// TIA Portal project "pidverdaero" (V16)
// Vorlageprojekt für das Buch mit Zielsystem S7-1200

(* hardware
DEVICE "S7-1200-Station_1"  S7-1200 Station
   slot 0: "Baugruppenträger_0"  Rack  V1.0
   slot 1: "PLC_1"  CPU 1211C DC/DC/DC  6ES7 211-1AE40-0XB0  V4.1
   slot 3: "AQ 1x12BIT_1"  AQ1 signal board  6ES7 232-4HA30-0XB0  V1.0
DEVICE "HMI_1"  TP900 Comfort
   slot 0: "HMI_1"  TP900 Comfort  6AV2 124-0JC01-0AX0  16.0.0.0
   slot 1: "HMI_RT_1"  TP900 Comfort  6AV2 124-0JC01-0AX0  16.0.0.0
   slot 5: "HMI_1.IE_CP_1"  PROFINET Interface  16.0.0.0
      slot 1: "Interfaz PROFINET_1"  PROFINET Interface
         slot 1: "Port_1"  Port
         slot 2: "Port_2"  Port
   slot 7: "HMI_1.MPI/DP_CP_1"  MPI/DP Interface  16.0.0.0
*)

// ===== PLC "PLC_1"  CPU 1211C DC/DC/DC =====

VAR_GLOBAL   // PLC tag table "Standard-Variablentabelle"
   "l2" AT %MD40 : Real;
   "l1" AT %MD44 : Real;
   "Kd1" AT %MD0 : Real;
   "Kd2" AT %MD4 : Real;
   "x1e" AT %MD8 : Real;
   "x2e" AT %MD12 : Real;
   "ue" AT %MD16 : Real;
   "u_min" AT %MD20 : Real;
   "u_max" AT %MD24 : Real;
   "z1" AT %MD28 : Real;
   "z2" AT %MD32 : Real;
   "delta_u" AT %MD36 : Real;
   "u_out" AT %MD48 : Real;
   "v1" AT %QD4 : Real;
   "AI_L1" AT %ID4 : Real;
   "AI_L2" AT %ID8 : Real;
   "AO_u" AT %QD0 : Real;
   "x1_hat" AT %MD52 : Real;
   "x2_hat" AT %MD56 : Real;
   "L1_1" AT %MD60 : Real;
   "L1_2" AT %MD64 : Real;
   "L2_1" AT %MD68 : Real;
   "L2_2" AT %MD72 : Real;
   "y1_dev" AT %MD76 : Real;
   "y2_dev" AT %MD80 : Real;
   "x1_hat_dev" AT %MD84 : Real;
   "x2_hat_dev" AT %MD88 : Real;
   "corr1" AT %MD92 : Real;
   "corr2" AT %MD96 : Real;
   "A11" AT %MD100 : Real;
   "A12" AT %MD104 : Real;
   "A21" AT %MD108 : Real;
   "A22" AT %MD112 : Real;
   "B1" AT %MD116 : Real;
   "B2" AT %MD120 : Real;
   "resid1" AT %MD124 : Real;
   "resid2" AT %MD128 : Real;
   "pred1" AT %MD132 : Real;
   "pred2" AT %MD136 : Real;
   "corr_term1" AT %MD140 : Real;
   "corr_term2" AT %MD144 : Real;
   "err1" AT %MD148 : Real;
   "err2" AT %MD152 : Real;
   "start" AT %I60.0 : Bool;
   "pid11" AT %Q8.0 : Bool;
   "pid22" AT %Q8.1 : Bool;
   "Kp" AT %MD156 : Real;
   "Ki" AT %MD160 : Real;
   "Kd" AT %MD164 : Real;
   "Ts" AT %MD168 : Real;
   "SetPoint" AT %MD172 : Real;
   "error" AT %MD176 : Real;
   "P_term" AT %MD180 : Real;
   "I_term" AT %MD184 : Real;
   "I_prev" AT %MD188 : Real;
   "D_term" AT %MD192 : Real;
   "error_prev" AT %MD196 : Real;
   "u_raw" AT %MD200 : Real;
END_VAR

DATA_BLOCK "OnOff_DB"   // DB2
{ S7_Optimized_Access := 'TRUE' }
VERSION : 0.1
// stored: InstanceOfName OnOff
"OnOff"
BEGIN
END_DATA_BLOCK

DATA_BLOCK "OnOff_DB2"   // DB4
{ S7_Optimized_Access := 'TRUE' }
VERSION : 0.1
// stored: InstanceOfName OnOff
"OnOff"
BEGIN
END_DATA_BLOCK

DATA_BLOCK "OnOff_DB_1"   // DB5
{ S7_Optimized_Access := 'TRUE' }
VERSION : 0.1
// stored: InstanceOfName OnOff
"OnOff"
BEGIN
END_DATA_BLOCK

DATA_BLOCK "I"   // DB6
{ S7_Optimized_Access := 'TRUE' }
VERSION : 0.1
// stored: InstanceOfName lqg1
"lqg1"
BEGIN
END_DATA_BLOCK

// folder: System blocks/Program resources

DATA_BLOCK "IEC_Timer_0_DB"   // DB1
{ S7_Optimized_Access := 'TRUE' }
AUTHOR : Simatic
FAMILY : IEC
NAME : IEC_TMR
VERSION : 1.0
// stored: InstanceOfName IEC_TIMER
"IEC_TIMER"
BEGIN
END_DATA_BLOCK

// folder: (top level)

FUNCTION_BLOCK "OnOff"   // FB1, SCL
{ S7_Optimized_Access := 'TRUE' }
VERSION : 0.1
BEGIN
   // ==============================
   // 0) PARÁMETROS PID (BALANCEADO)
   // ==============================
   // Ganancias calculadas con pidtune (Robustez 60deg)
   "Kp" := 2.9222;
   "Ki" := 0.0231;
   "Kd" := 32.0832;

   // Tiempo de muestreo (Debe ser igual al Cyclic Interrupt, ej. 0.05s)
   "Ts" := 0.05;

   // Referencia (Set Point) - A donde quieres que llegue el agua
   "SetPoint" := 2.0;

   // Límites del Actuador
   "u_min" := 0.0;
   "u_max" := 10.0;

   // ==============================
   // 1) LECTURA Y ESCALADO (IGUAL AL LQG)
   // ==============================

   "l1" := ("l1" * 0.9) + (("AI_L1" * 0.3) * 0.1);
   "l2" := "AI_L2" * 0.3;

   // Cálculo de caudal (Solo para monitoreo)
   "v1" := 4.073 * SQRT("l2");

   // ==============================
   // 2) CÁLCULO DEL ERROR
   // ==============================

   // Error actual = Lo que quiero - Lo que tengo
   "error" := "SetPoint" - "l1";

   // ==============================
   // 3) ALGORITMO PID
   // ==============================

   // --- TÉRMINO PROPORCIONAL (P) ---
   "P_term" := "Kp" * "error";

   // --- TÉRMINO INTEGRAL (I) ---
   // Acumula el error: I_nuevo = I_viejo + (Ki * error * Tiempo)
   // "I_prev" debe ser variable STATIC (Memoria)
   "I_term" := "I_prev" + ("Ki" * "error" * "Ts");

   // --- TÉRMINO DERIVATIVO (D) ---
   // Velocidad del error: D = Kd * (error - error_anterior) / Tiempo
   // "error_prev" debe ser variable STATIC (Memoria)
   "D_term" := "Kd" * ("error" - "error_prev") / "Ts";

   // --- SUMA TOTAL ---
   "u_raw" := "P_term" + "I_term" + "D_term";

   // ==============================
   // 4) SATURACIÓN Y ANTI-WINDUP
   // ==============================

   IF "u_raw" > "u_max" THEN
       "u_out" := "u_max";
       "I_term" := "I_prev"; // Congelar Integral

   ELSIF "u_raw" < "u_min" THEN
       "u_out" := "u_min";
       "I_term" := "I_prev"; // Congelar Integral

   ELSE
       "u_out" := "u_raw";
       "I_prev" := "I_term"; // Guardar Integral nueva
   END_IF;

   // ==============================
   // 5) ACTUALIZACIÓN DE MEMORIAS
   // ==============================
   // Guardamos el error actual para usarlo como "pasado" en el siguiente ciclo
   "error_prev" := "error";

   // ==============================
   // 6) SALIDA AL ACTUADOR
   // ==============================
   "AO_u" := "u_out";
END_FUNCTION_BLOCK

FUNCTION_BLOCK "lqg1"   // FB2, SCL
{ S7_Optimized_Access := 'TRUE' }
VERSION : 0.1
BEGIN
   // ==========================================
   // 1. PARÁMETROS (Tus Ganancias Altas)
   // ==========================================
   "Kp" := 4.1326;
   "Ki" := 0.0461;
   "Kd" := 82.0658;

   "Ts" := 0.05;      // Tiempo de ciclo
   "SetPoint" := 1.0; // Referencia (1 metro)
   "u_min" := 0.0;
   "u_max" := 10.0;

   // ==========================================
   // 2. LECTURA Y FILTRO (EN UNA SOLA LÍNEA)
   // ==========================================

   // Truco: Usamos "l1" para guardar el valor filtrado. 
   // 0.9 = Memoria (Suavidad) | 0.1 = Lectura Nueva (Sensor)
   // ESTO ELIMINA EL RUIDO SIN CREAR VARIABLES NUEVAS
   "l1" := ("l1" * 0.9) + (("AI_L1" * 0.3) * 0.1);

   // Lectura Tanque 2 (Solo visual, sin filtro)
   "l2" := "AI_L2" * 0.3;
   "v1" := 4.073 * SQRT("l2");

   // ==========================================
   // 3. CÁLCULO DEL ERROR
   // ==========================================
   "error" := "SetPoint" - "l1";

   // ==========================================
   // 4. ALGORITMO PID (ESTÁNDAR)
   // ==========================================

   // -- PROPORCIONAL --
   "P_term" := "Kp" * "error";

   // -- INTEGRAL (ACUMULATIVA) --
   // "I_prev" DEBE SER STATIC (Memoria)
   "I_term" := "I_prev" + ("Ki" * "error" * "Ts");

   // -- DERIVATIVO (VELOCIDAD) --
   // "error_prev" DEBE SER STATIC (Memoria)
   "D_term" := "Kd" * ("error" - "error_prev") / "Ts";

   // -- SUMA TOTAL --
   "u_raw" := "P_term" + "I_term" + "D_term";

   // ==========================================
   // 5. SATURACIÓN Y ANTI-WINDUP
   // ==========================================

   IF "u_raw" > "u_max" THEN
       "u_out" := "u_max";
       "I_term" := "I_prev"; // Congelar Integral

   ELSIF "u_raw" < "u_min" THEN
       "u_out" := "u_min";
       "I_term" := "I_prev"; // Congelar Integral

   ELSE
       "u_out" := "u_raw";
       "I_prev" := "I_term"; // Guardar Integral nueva
   END_IF;

   // ==========================================
   // 6. GUARDAR MEMORIA
   // ==========================================
   "error_prev" := "error"; // Guardar error para la derivada del siguiente ciclo

   // ==========================================
   // 7. SALIDA FÍSICA
   // ==========================================
   "AO_u" := "u_out";
END_FUNCTION_BLOCK

FUNCTION "MHJ-PLC-Lab-Function-S71200" : Void   // FC9000, SCL
{ S7_Optimized_Access := 'TRUE' }
VERSION : 0.1
   VAR_TEMP
      rdTimeReturn : Int;
      outputTime : DTL;
      SyncVal : Byte;
      forVal : Int;
      forVal_2 : Int;
      Value : Byte;
   END_VAR
   VAR CONSTANT
      CompVal : Byte := 16#34;
      Value_01 : Byte := 16#11;
      Value_01_DW : DWord := 16#A165_D992;
      Value_02_DW : DWord := 16#58BE_4401;
   END_VAR
BEGIN

   #Value:=PEEK(area := 16#82,
        dbNumber := 0,
        byteOffset := 511);
   #Value := #Value + 1;

   POKE(area := 16#82,
        dbNumber := 0,
        byteOffset := 511,
        value := #Value);

   POKE(area:=16#81,
        dbNumber:=0,
        byteOffset:=1016,
        value:=#Value_01_DW);
   POKE(area := 16#81,
        dbNumber := 0,
        byteOffset := 1020,
        value := #Value_02_DW);

   POKE(area := 16#81,
        dbNumber := 0,
        byteOffset := 511,
        value := B#16#00);

   FOR #forVal := 0 TO 120 DO
       FOR #forVal_2:=0 TO 10 DO
           #rdTimeReturn:=RD_SYS_T(#outputTime);
           #rdTimeReturn := WR_SYS_T(#outputTime);
           #rdTimeReturn := RD_SYS_T(#outputTime);
           #rdTimeReturn := WR_SYS_T(#outputTime);
       END_FOR;
       #SyncVal:= PEEK(area := 16#81,
                      dbNumber := 0,
                      byteOffset := 511);
       IF #SyncVal = #CompVal THEN
          GOTO M_1;
       END_IF;
   END_FOR;
   RETURN;

   M_1:
   POKE(area := 16#81,
        dbNumber := 0,
        byteOffset := 511,
        value := B#16#0);
END_FUNCTION

ORGANIZATION_BLOCK "Main"   // OB1, LAD, ProgramCycle
TITLE = "Main Program Sweep (Cycle)"
{ S7_Optimized_Access := 'TRUE' }
VERSION : 0.1
   VAR_INPUT
      Initial_Call : Bool;   // Initial call of this OB
      Remanence : Bool;   // =True, if remanent data are available
   END_VAR
   VAR_TEMP   // added for the SCL form of the ladder/FBD networks
      _w1 : Bool;
      _w2 : Bool;
   END_VAR
BEGIN

REGION Network 1: Konnektierungsbaustein für PLC-Lab
   // Im Netzwerk 1 wird der Konnektierungsbaustein für PLC-Lab aufgerufen.
   // Dieser Aufruf darf nicht entfernt werden!
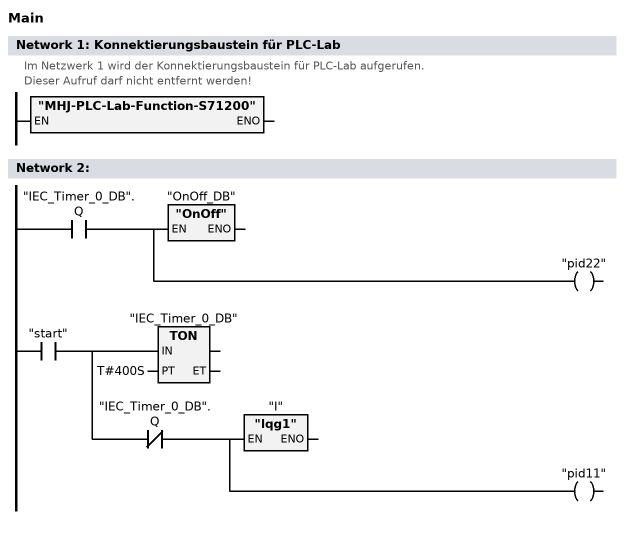
   RUNG wire#powerrail
      "MHJ-PLC-Lab-Function-S71200"()
   END_RUNG
   // the same network as SCL:
   "MHJ-PLC-Lab-Function-S71200"();
END_REGION

REGION Network 2
   #_w1 := "IEC_Timer_0_DB".Q;
   IF #_w1 THEN
       "OnOff_DB"();   // "OnOff"
   END_IF;
   "pid22" := #_w1;
   "IEC_Timer_0_DB".TON(IN := "start", PT := T#400S);
   #_w2 := "start" AND NOT "IEC_Timer_0_DB".Q;
   IF #_w2 THEN
       "I"();   // "lqg1"
   END_IF;
   "pid11" := #_w2;
END_REGION
END_ORGANIZATION_BLOCK

(* ===== HMI "HMI_RT_1" =====
system functions are stored by id; their names below are inferred from use
connection "HMI_Conexión_1": ETHERNET, S7_1200_OMS

HMI tags "Tabla de variables estándar"
   "Número_imagen_variable" : UInt, internal
   "l1" : Real = PLC l1 AT %MD44, 1 s
   "l2" : Real = PLC l2 AT %MD40, 1 s
   "AO_u" : Real = PLC AO_u AT %QD0, 1 s

screen "Imagen raíz" 800x420, template "Plantilla_1"
   on GenerateScreen: SetTag("Número_imagen_variable", 1)
   TrendView "Visor de curvas_1" at 8,5 size 787x351

Template "Plantilla_1" 800x420
   Button "Exit" at 720,360 size 78x58; TextOff 'Exit'; PictureOff "ExitRuntime_TP900_Comfort_TR"; PictureOn "ExitRuntime_TP900_Comfort_TR"
      on Release: StopRuntime(0)
   Button "Template_Button" at 640,360 size 78x58; TextOff 'Text'
   Button "Template_Button_1" at 560,360 size 78x58; TextOff 'Text'
   Button "Template_Button_2" at 480,360 size 78x58; TextOff 'Text'
   Button "Template_Button_3" at 400,360 size 78x58; TextOff 'Text'
   Button "Template_Button_4" at 321,360 size 78x58; TextOff 'Text'
   Button "Template_Button_5" at 241,360 size 78x58; TextOff 'Text'
   Button "Template_Button_6" at 161,360 size 78x58; TextOff 'Text'
   Button "Template_Button_7" at 81,360 size 78x58; TextOff 'Text'
   Button "Start screen" at 1,360 size 78x58; TextOff 'Start screen'; PictureOff "NavigateHome_TP900_Comfort_TR"; PictureOn "NavigateHome_TP900_Comfort_TR"
      on Release: ActivateScreen("Imagen raíz", 0)
*)